Fanuc KAREL source: kd00019.KL

-- PROVISIONAL review KL for V770-1; original PC SHA256 973c24aa6d4bca90701eaef9c61b8b0653396c3922e814eea720cbde2738c8d3
-- Incomplete behavior may be omitted. Consult companion uncertainty JSON. Do not deploy.
PROGRAM KD00019
%NOLOCKGROUP
VAR
  I : INTEGER
  J : INTEGER
  B : BOOLEAN
  R : REAL
  S : STRING[80]
-- UNRESOLVED_DECL REC type=001100
BEGIN
  -- UNRESOLVED_PC offsets 5-16; opcodes 9D,22,32,35
  -- UNRESOLVED_PC offsets 26-48; opcodes 22,32,34,9D,52,22,32,35
  -- UNRESOLVED_PC offsets 58-62; opcodes 7F
END KD00019
